TYPE "AnalogSens_HmiData"
VERSION : 0.1
// Block: AnalogSens_HmiData
   STRUCT
      PbPreset : Bool;
      PresetValue : LReal;
      PresetFdback : LReal;
   END_STRUCT;

END_TYPE
